(*
SPDX-FileCopyrightText: © 2026 Oleksandr Tiutyk <trofimich@gmail.com>
SPDX-License-Identifier: MIT
License: https://opensource.org/license/mit
*)

(*!
<summary>Identifies the active phase of a running task.</summary>
<description>
Acquisition, processing, stopping and release are diagnostic substates, not independent scheduling tasks.
Interpret them only while TASK_STATE is RUNNING.
</description>
*)
{attribute 'qualified_only'}
{attribute 'strict'}
{attribute 'to_string'}
TYPE TASK_RUNNING_SUBSTATE :
(
	//! <summary>Acquire the resource before ordinary work.</summary>
	RESOURCE_ACQUIRING := 0,
	//! <summary>Advance ordinary work unless cancellation is pending.</summary>
	PROCESSING,
	//! <summary>Advance the terminal resource-release attempt.</summary>
	RESOURCE_RELEASING,
	//! <summary>Finish active work for any stop reason before resource release.</summary>
	STOPPING
);
END_TYPE

(* stored: Version 1.1.0.1
   DUT TASK_RUNNING_SUBSTATE: Id {97e9448b-3744-40b9-9500-a0e82cc27ef6} *)
